FUNCTION_BLOCK FB_CreatePingMessage_Test EXTENDS TcUnit.FB_TestSuite
VAR_INPUT
END_VAR
VAR_OUTPUT
END_VAR
VAR
END_VAR

Nominal();

METHOD Nominal : REFERENCE TO FB_Test
VAR_INPUT
END_VAR
VAR
	pJsonBuffer : POINTER TO STRING(255);
	stMsg : _ST_SiftMessage;
	stErr : ST_SiftError;
	sExpectedJson : STRING(255) := '{"endpoint":"ping","data":{}}';
END_VAR
// Test creating a nominal ping message.
TEST('CreatePingMessage Nominal');

stErr := _F_CreatePingMessage(stMsg := stMsg);
								
AssertFalse(stErr.bError, Message := 'error creating ping message');

pJsonBuffer := ADR(stMsg.aData);
AssertEquals_STRING(Expected := sExpectedJson, 
				    Actual := pJsonBuffer^, 
				    Message := 'bad ping message was created');

TEST_FINISHED();
END_METHOD

END_FUNCTION_BLOCK

(* stored: Version 1.1.0.1
   POU FB_CreatePingMessage_Test: Id {cff0359a-aba1-453d-9fa5-12970330a1d2}, SpecialFunc None
   Method Nominal: Id {154f45f7-bbc0-4aa4-b76b-cac0a0fe646a} *)
